// TIA Portal V18 export
ORGANIZATION_BLOCK "17-Cabin Movement"   // OB124, LAD, ProgramCycle
TITLE = "Main Program Sweep (Cycle)"
{ S7_Optimized_Access := 'TRUE' }
VERSION : 0.1
// stored: AutoNumber true, IsIECCheckEnabled false, SetENOAutomatically false
   VAR_INPUT
      Initial_Call : Bool;   // Initial call of this OB
      Remanence : Bool;   // =True, if remanent data are available
   END_VAR
   VAR_TEMP
      "Cab Angle NormScale" : Real;
   END_VAR
   VAR_TEMP   // added for the SCL form of the ladder/FBD networks
      _w1 : Bool;
   END_VAR
BEGIN

REGION Network 1: Cab Movement
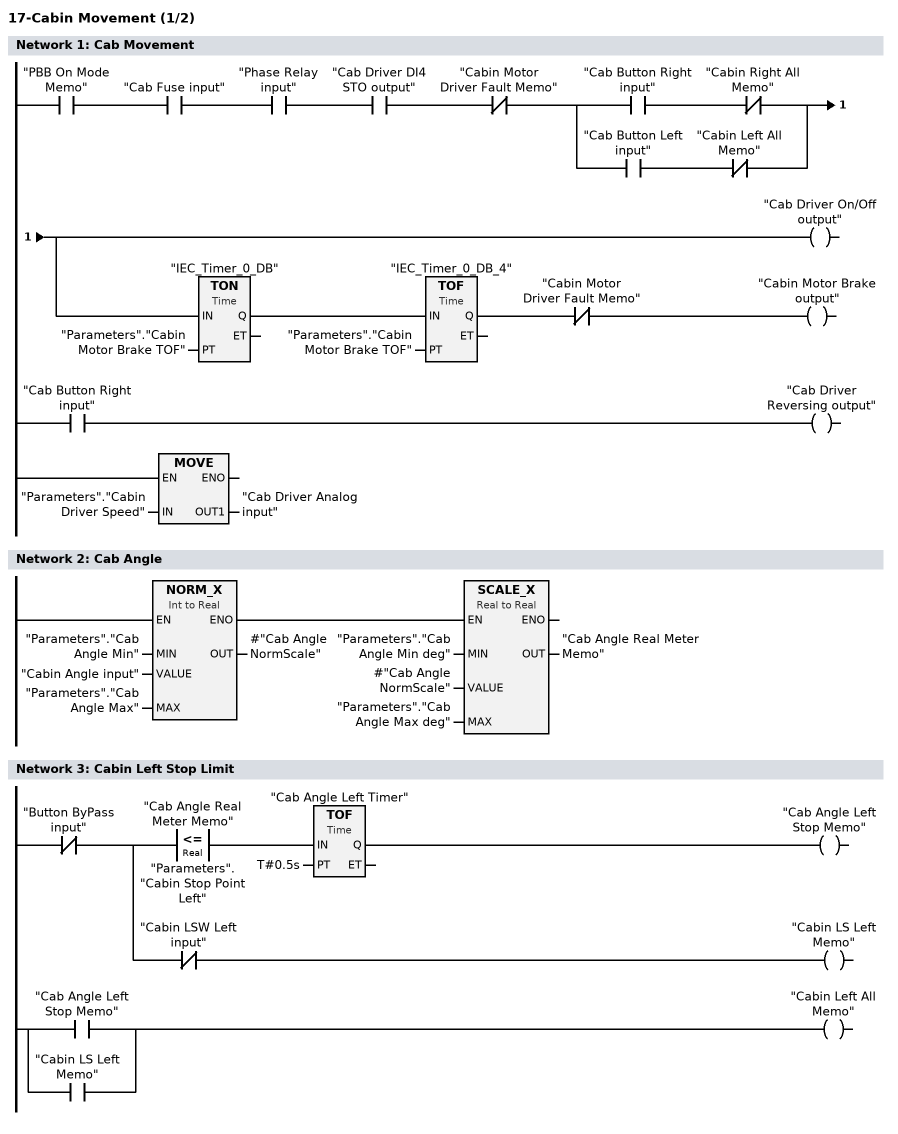
   RUNG wire#powerrail
      Contact( "PBB On Mode Memo" )
      Contact( "Cab Fuse input" )
      Contact( "Phase Relay input" )
      Contact( "Cab Driver DI4 STO output" )
      I_Contact( "Cabin Motor Driver Fault Memo" )
      wire#w1
      Contact( "Cab Button Right input" )
      I_Contact( "Cabin Right All Memo" )
      wire#w2
      Coil( "Cab Driver On/Off output" )
   END_RUNG
   RUNG wire#w1
      Contact( "Cab Button Left input" )
      I_Contact( "Cabin Left All Memo" )
   END_RUNG wire#w2
   RUNG wire#w2
      { S7_Templates := "time_type := Time" } "IEC_Timer_0_DB".TON(pt := "Parameters"."Cabin Motor Brake TOF", et =>)
      { S7_Templates := "time_type := Time" } "IEC_Timer_0_DB_4".TOF(pt := "Parameters"."Cabin Motor Brake TOF", et =>)
      I_Contact( "Cabin Motor Driver Fault Memo" )
      Coil( "Cabin Motor Brake output" )
   END_RUNG
   RUNG wire#powerrail
      Contact( "Cab Button Right input" )
      Coil( "Cab Driver Reversing output" )
   END_RUNG
   RUNG wire#powerrail
      Move(in := "Parameters"."Cabin Driver Speed", out1 => "Cab Driver Analog input")
   END_RUNG
   // the same network as SCL:
   "Cab Driver On/Off output" := "PBB On Mode Memo" AND "Cab Fuse input" AND "Phase Relay input" AND "Cab Driver DI4 STO output" AND NOT "Cabin Motor Driver Fault Memo" AND (("Cab Button Right input" AND NOT "Cabin Right All Memo") OR ("Cab Button Left input" AND NOT "Cabin Left All Memo"));
   "IEC_Timer_0_DB".TON(IN := "Cab Driver On/Off output", PT := "Parameters"."Cabin Motor Brake TOF");
   "IEC_Timer_0_DB_4".TOF(IN := "IEC_Timer_0_DB".Q, PT := "Parameters"."Cabin Motor Brake TOF");
   "Cabin Motor Brake output" := "IEC_Timer_0_DB_4".Q AND NOT "Cabin Motor Driver Fault Memo";
   "Cab Driver Reversing output" := "Cab Button Right input";
   "Cab Driver Analog input" := "Parameters"."Cabin Driver Speed";
END_REGION

REGION Network 2: Cab Angle
   RUNG wire#powerrail
      { S7_Templates := "[SrcType := Int, DestType := Real]" } Normalize(min := "Parameters"."Cab Angle Min", value := "Cabin Angle input", max := "Parameters"."Cab Angle Max", out => #"Cab Angle NormScale")
      { S7_Templates := "[SrcType := Real, DestType := Real]" } Scale(min := "Parameters"."Cab Angle Min deg", value := #"Cab Angle NormScale", max := "Parameters"."Cab Angle Max deg", out => "Cab Angle Real Meter Memo")
   END_RUNG
   // the same network as SCL:
   #"Cab Angle NormScale" := NORM_X(MIN := "Parameters"."Cab Angle Min", VALUE := "Cabin Angle input", MAX := "Parameters"."Cab Angle Max");
   "Cab Angle Real Meter Memo" := SCALE_X(MIN := "Parameters"."Cab Angle Min deg", VALUE := #"Cab Angle NormScale", MAX := "Parameters"."Cab Angle Max deg");
END_REGION

REGION Network 3: Cabin Left Stop Limit
   RUNG wire#powerrail
      I_Contact( "Button ByPass input" )
      wire#w1
      { S7_Templates := "SrcType := Real" } LE_Contact(in1 := "Cab Angle Real Meter Memo", in2 := "Parameters"."Cabin Stop Point Left")
      { S7_Templates := "time_type := Time" } "Cab Angle Left Timer".TOF(pt := T#0.5s, et =>)
      Coil( "Cab Angle Left Stop Memo" )
   END_RUNG
   RUNG wire#w1
      I_Contact( "Cabin LSW Left input" )
      Coil( "Cabin LS Left Memo" )
   END_RUNG
   RUNG wire#powerrail
      Contact( "Cab Angle Left Stop Memo" )
      wire#w2
      Coil( "Cabin Left All Memo" )
   END_RUNG
   RUNG wire#powerrail
      Contact( "Cabin LS Left Memo" )
   END_RUNG wire#w2
   // the same network as SCL:
   #_w1 := NOT "Button ByPass input";
   "Cab Angle Left Timer".TOF(IN := #_w1 AND ("Cab Angle Real Meter Memo" <= "Parameters"."Cabin Stop Point Left"),
                           PT := T#0.5s);
   "Cab Angle Left Stop Memo" := "Cab Angle Left Timer".Q;
   "Cabin LS Left Memo" := #_w1 AND NOT "Cabin LSW Left input";
   "Cabin Left All Memo" := "Cab Angle Left Stop Memo" OR "Cabin LS Left Memo";
END_REGION

REGION Network 4: Cabin Right Stop Limit
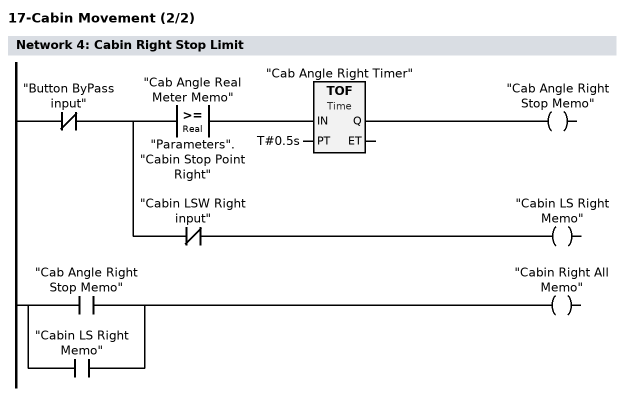
   RUNG wire#powerrail
      I_Contact( "Button ByPass input" )
      wire#w1
      { S7_Templates := "SrcType := Real" } GE_Contact(in1 := "Cab Angle Real Meter Memo", in2 := "Parameters"."Cabin Stop Point Right")
      { S7_Templates := "time_type := Time" } "Cab Angle Right Timer".TOF(pt := T#0.5s, et =>)
      Coil( "Cab Angle Right Stop Memo" )
   END_RUNG
   RUNG wire#w1
      I_Contact( "Cabin LSW Right input" )
      Coil( "Cabin LS Right Memo" )
   END_RUNG
   RUNG wire#powerrail
      Contact( "Cab Angle Right Stop Memo" )
      wire#w2
      Coil( "Cabin Right All Memo" )
   END_RUNG
   RUNG wire#powerrail
      Contact( "Cabin LS Right Memo" )
   END_RUNG wire#w2
   // the same network as SCL:
   #_w1 := NOT "Button ByPass input";
   "Cab Angle Right Timer".TOF(IN := #_w1 AND ("Cab Angle Real Meter Memo" >= "Parameters"."Cabin Stop Point Right"),
                           PT := T#0.5s);
   "Cab Angle Right Stop Memo" := "Cab Angle Right Timer".Q;
   "Cabin LS Right Memo" := #_w1 AND NOT "Cabin LSW Right input";
   "Cabin Right All Memo" := "Cab Angle Right Stop Memo" OR "Cabin LS Right Memo";
END_REGION
END_ORGANIZATION_BLOCK
